// TIA Portal V18 export
// export: Created 2026-01-09T11:23:23.9077287Z, ExportSetting WithDefaults, DisplayName Totally Integrated Automation Portal, DisplayVersion V18 Update 5, DisplayName TIA Portal Openness, DisplayVersion V18 Update 5, DisplayName TIA Portal Teamcenter Gateway, DisplayVersion V18, DisplayName TIA Portal Version Control Interface, DisplayVersion V18, DisplayName SINAMICS Startdrive Advanced, DisplayVersion V18 SP2 Update 1, DisplayName SINAMICS Startdrive G110M, G120, G120C, G120D, G120P, G115D, DisplayVersion V18 SP2 Update 1, DisplayName SINAMICS Startdrive G130, G150, S120, S150, SINAMICS MV, S210, G220, S200, DisplayVersion V18 SP2 Update 1, DisplayName STEP 7 Professional, DisplayVersion V18 Update 5, DisplayName STEP 7 Safety, DisplayVersion V18, DisplayName WinCC Professional, DisplayVersion V18 Update 5
Screen "02StationNumber"  1280x800, Number=2, Template=11GMT
  on GenerateScreen: Loading(); SetBit(Tag := NormalON); ResetBit(Tag := NormalOFF); VBCom(Index := 5); LoadIO(); IOVisual(Funcode := 100, SubFuncode := 0)
  ScreenLayer 
    SymbolicIOField "seaText1" at 131,72 size 1146x65  CountVisibleItems=3, Mode=Output, OnValue=1, StyleItem=sltDeepBold22, TextList=XXXXX_PanelTextlist, TextOff="OP010", TextOn="OP010"
      ProcessValue := Sys_VersionManagement_HMIPageID
    TextField "文本域_7" at 151,141 size 367x37  Text="站介绍 / Station Introduction / Úvod do stanice"
    GraphicView "图形视图_1" at 154,195 size 677x508  Picture=图形_43
    Button "btnMenu1_1" at 0,70 size 128x75  Mode=Text, PictureOff=SS_00_000_HomeSmall, StyleItem=BtnActive18, TextOff="工位号 / Station Number / Stanica Číslo"
      on Release: ActivateScreen(Screen name := , Object number := 0); SetTag(Tag := Sys_VersionManagement_HMIPageID, Value := 2)
    TextField "文本域_2" at 843,201 size 428x124  Text="此工站为组装工站，把Ring1、Ring2、Shaft Magnet、通过压装、涂胶、固化涂胶等工艺装 配到一起，产出初步转子产品。 / This workstation is an assembly station whereRing1, Ring2, and Shaft Magnet are assembled together through pressing, gluing, and curingprocesses to produce preliminary rotor products. / Táto pracovná stanica je montážna stanica , kde sa Ring1, Ring2 a Shaft Magnet montujú spolu pomocou lisovania, nanášania lepidla a vytvrdzovania lepidla, čím vzniká počiatočný rotorový produkt."
